{attribute 'Tc2GvlVarNames'}
VAR_CONFIG
END_VAR

(* stored: Version 1.1.0.1, ProductVersion 3.1.0.36
   GVL Variablen_Konfiguration: Id {f965ba7c-3df1-4141-9c7c-deae8c5059d5} *)
